Staubli VAL3: parkEndProgram.pgx

program parkEndProgram()
  local jointRs jPos
begin
  if bEndProgram==true
    call print("end program, put robot into safe state")

    statusDoAirex       = colorError
    statusCleanupChuck1 = colorError
    statusCleanupChuck2 = colorError
    statusDoModules     = colorError

    jPos = herej()
    call print("end program: stopMove at here.z = "  + toString("6.3", jPos.j3))
    delay(1)
    stopMove()

   // jPos = herej()
    call print("end program: resetMotion at here.z = "  + toString("6.3", jPos.j3))
    delay(1)
    resetMotion()


    // -- move up to safe z position from wherever you are
    jPos.j3 = 70
    call print("end program: move up")
    movej(jPos, tTool, mSlow)
    waitEndMove()

    // -- move over end of foil, deposit anything connected
    call print("end program: move to appro(parkEndPoint, trZsafe)")
    movej(appro(parkEndPoint, trZsafe), tTool, mNomSpeed)
    waitEndMove()
    call print("end program: move to appro(parkEndPoint, trZero)")
    movej(appro(parkEndPoint, trZero), tTool, mSlow)
    waitEndMove()
    call print("end program: drop tool")
    switchMagnet = false
    switchVac0   = false
    switchVac1   = false
    delay(1)

    // -- move up
    call print("end program: move up")
    movej(appro(parkEndPoint, trZsafe), tTool, mNomSpeed)
    waitEndMove()

    // -- move to normal rest position
    call print("end program: move to normal rest position")
    movej(jInitialPosition, tTool, mFast)
    waitEndMove()
    resetMotion()

    //taskKill("doAirexTask")
    //taskKill("doModulesTask")
    //taskKill("doGlueGlass")

    bEndProgram = false
    disablePower()
    call print("program ended, now what?")
  endIf

end
